(* CODESYS project CtaAppPid_2.0.0.0.library
   Description: PID Library der CTA
   Version: 2.0.0.0
   Title: CtaAppPid
   Author: SIS
   DocFormat: reStructuredText
   Placeholder: CtaAppPid
   LanguageModelAttribute: qualified-access-only
   DefaultNamespace: CtaAppPid
   CompiledLibraryCompatibilityVersion: CODESYS V3.5 SP16 Patch 3
   Company: CTA

Project tree, tasks and I/O mapping:
  libraries: CtaSysConfig, 2.0.0.0 (CTA); CtaAppTime, 1.0.0.1 (CTA); VisuSymbols, 4.5.0.0 (System); CtaVisSymbols, 2.0.0.0 (CTA); Standard, 3.5.18.0 (System); CtaAppInfluxLog, 1.0.0.1 (CTA); CtaVisHelp, 1.0.0.0 (CTA); CtaVisUser, 1.0.0.0 (CTA)
  40 Visualizations/
    visualisation popUpPID
    visualisation visPID
  30 Program Organization Units/
    function block fbPid [ST]: actConfigFile, actTrendLog, proInvert
  00000000-0000-0000-0000-000000000000|D:\CoDeSys\LibrariesV3\trunk\Intern\CAA\CAA Template\3.4.0.0 draft\Placeholder.xml
  00000000-0000-0000-0000-000000000000|D:\CoDeSys\LibrariesV3\trunk\Intern\CAA\CAA Template\3.2.0.3 draft\Prefix.pdf
  00000000-0000-0000-0000-000000000000|D:\CoDeSys\LibrariesV3\trunk\Intern\CAA\CAA Template\3.5.2.0 draft\Placeholder.xml
  20 Structs/
    data type scParameter
  50 Images/
  10 Documenation/
    global variables VersionHistory
    global variables readMe
  21 Interface/
  11 Library Parameter/
  12 Konstanten/
  60 Textlisten/
  13 Globale Variablen/
  text list GlobalTextList
*)

// 20 Structs/scParameter
TYPE scParameter :
    STRUCT
        fbrDeadBand     	:   CtaSysConfig.fbREAL;   // Dead Band
        fbrBand         	:   CtaSysConfig.fbREAL;   // Bereich in den Integriert wird in REAL
        fbrTn           	:   CtaSysConfig.fbREAL;   // Integrations Zeit in REAL 60.0 = 60.0 SEC
        fbrTv           	:   CtaSysConfig.fbREAL;   // Differential Zeit in REAL 60.0 = 60.0 SEC       
        fbxInvert			:   CtaSysConfig.fbBOOL;   // Regelverhalten Invertieren 
		fbxEnTrendlog		:	CtaSysConfig.fbBOOL;
    END_STRUCT
END_TYPE

// 10 Documenation/VersionHistory
(* 

.. image:: ../../Images/CTA_Logo.jpg
   :align: right
   :width: 15% 

**Vorlage**   


============ =========== =========== ============================================
**Date**     **Version** **Author**  **Change**
------------ ----------- ----------- --------------------------------------------
04.03.2021   0.0.0.0     SIS         Vorlage erstellt

============ =========== =========== ============================================


*)
VAR_GLOBAL
    stInfo : STRING:= '0.0.0.0, Vorlage, CTA';
END_VAR

// 10 Documenation/readMe
(*

**ReadMe**
 
 |  **Empfehlung**
 |
 |	Bibliothek CtaAppPid zur implementierung eine PID- Reglers.
 |  Instanzieren Sie den CtaAppPid.fbPid in ihrem Funktionsbaustein oder POU beispielsweise als fbPidX(Komponente)Y. (X = Nr des Reglers; Komponente z.B Pumpe, Antrieb oder Ventilator; Y = Nr der Komponente) 
 |  Deklarieren Sie die Struktur Variable welche als Parameter und zur ansteuerung dienen wie im Code beispiel.
 |  
 |  *Beispiel* 

+-----------------------+---------------------------------------------------------------------------------------------------------------------------------------------------------------------------------------------------------------------------------------------------------------------------------------------------------------------------------------------------------------------------------------------------------------------------------------+
| Beschreibung          |  Code                                                                                                                                                                                                                                                                                                                                                                                                                                 |
+=======================+=======================================================================================================================================================================================================================================================================================================================================================================================================================================+
| Pou oder SmFb         | .. code-block:: codesys                                                                                                                                                                                                                                                                                                                                                                                                               |
|                       |                                                                                                                                                                                                                                                                                                                                                                                                                                       |
|                       |	// Deklaration als VAR im POU oder dem selbsterstellten Funktionsbaustein                                                                                                                                                                                                                                                                                                                                                       	|
|                       |   VAR   																																																																																																								|
|						|	    (*PID*)																																																	 																																																						|
|						|		fbPid1Pumpe1			: CtaAppPid.fbPid;                                                                                                                                                                                                                                                                                                                                                              						|
|                       | 		fbPid2Pumpe1			: CtaAppPid.fbPid;																																																																																														|
| 						|	END_VAR                                                                                                                                                                                                                                                                                                                                                                                                                         	|
+-----------------------+---------------------------------------------------------------------------------------------------------------------------------------------------------------------------------------------------------------------------------------------------------------------------------------------------------------------------------------------------------------------------------------------------------------------------------------+
| Code für Init         | .. code-block:: codesys                                                                                                                                                                                                                                                                                                                                                                                                               |
|                       |   																																																																																																									|
| 						|	// Kopieren des nachfolgenden Codes in eine Action zur Initialisierung der Parameter. Zum Beispiel actParameter.																																																																													|
|                       |	{region "Parameter Pid1Pumpe1"}                                                                                                                                                                                                                                                                                                                                                                                                     |
| 						|		(*Basis*)																																																																																																						|
|						|		fbPid1Pumpe1.scParameter.fbrDeadBand               		(_wertInit :=   0.0									, _minInit :=   	, _maxInit := 		);		//P1 Totband																																																														|
|						|		fbPid1Pumpe1.scParameter.fbrBand						(_wertInit :=   0.0									, _minInit :=   	, _maxInit := 		);		//P2 P- Band																																																														|
|						|		fbPid1Pumpe1.scParameter.fbrTn							(_wertInit :=   0.0									, _minInit :=   	, _maxInit := 		);		//P3 Nachstellzeit																																																													|
|						|		fbPid1Pumpe1.scParameter.fbrTv							(_wertInit :=   0.0									, _minInit :=   	, _maxInit := 		);		//P4 Vorhaltezeit																																																													|
|						|		fbPid1Pumpe1.scParameter.fbxInvert						(_wertInit := FALSE																			);		//P5 Regler Invertierung																																																											|
|						|	{endregion}                                                                                                                                                      																																																																	| 
+-----------------------+---------------------------------------------------------------------------------------------------------------------------------------------------------------------------------------------------------------------------------------------------------------------------------------------------------------------------------------------------------------------------------------------------------------------------------------+
*)                                                                                                                                                                                                                                                                                                                                                                                                                                                               
 VAR_GLOBAL                                                                                                                                                                                                                                                                                                                                                                                                                                                      
    xReadMeDone              :   BOOL;                                                                                                                                                                                                                                                                                                                                                                                                                           
END_VAR

// 30 Program Organization Units/fbPid
//*******************************************************************************************************************************************************************************************************************************************//
//  Author:         SIS                                                                           																																			 //
//  Version:        1.0.0.0		                                                                      																																		 //
//  Beschreibung:   PID Regler                                                                   																																			 //
//  rIntegral =(((rAct-rSoll)/rBand*2000)/(rTn) *(rCycleTime) + rIntegral)     																										                                                	     //
//  rProp = ((rAct-rSoll)/rBand*2000)                                          																						 				                                                		 //
//  Regler Wert = ( rProp + rIntegral + rDiff)                                 																										                                                	  	 //
//*******************************************************************************************************************************************************************************************************************************************//
{attribute 'reflection'} 
FUNCTION_BLOCK fbPid 
//===========================================================================================================================================================================================================================================//
//  Variabeln Deklaration  Input                                                                  																																			 //
//===========================================================================================================================================================================================================================================//
VAR_INPUT   
    xEn                         :   BOOL;   // regler Freigabe                   
    rAct                        :   REAL;   // regelwert X in REAL
    rSoll                       :   REAL;   // Regelwert W in REAL     
    stPhysikalischeEinheit      :   STRING[5];
END_VAR
//===========================================================================================================================================================================================================================================//
//  Variabeln Deklaration  Output                                                                																																			 //
//===========================================================================================================================================================================================================================================//
VAR_OUTPUT                     
    rY              :   REAL;   // Stellgrösse Y
END_VAR
VAR
    {attribute 'instance-path'} 
    {attribute 'noinit'} 
    stInstanzName   :   STRING;
    xInitDone       :   BOOL;                                   // Inititalisierung Abgeschlossen
    scParameter     :   scParameter;
    xSimulation     :   BOOL;                                   // Simultion Aktiv
    xSimOn          :   BOOL;                                   // Simulationstrigger On
    xSimOff         :   BOOL;                                   // Simulationstrigger Off    
    rSollSim        :   REAL;                                   // Simulations Regelwert W in REAL  
    rActSim         :   REAL;                                   // Simulation Regelwert X in REAL  
    rSollPid        :   REAL;                                   // Regelwert auf den Geregelt wird
    rActPid         :   REAL;                                   // Istwert auf den Geregelt wird 
    rProp           :   REAL;                                   // Proportional Wert
    rPropVisu       :   REAL;                                   // Proportional Wert für Visu Darstellung
    rIntegral       :   REAL;                                   // Integral Wert
    rDiff           :   REAL;                                   // Diferential Wert
    xCycleStart     :	BOOL;                                   // Startbefehl des Zyklus
    xCycleInterupt  :   BOOL;                                   // Zyklus ende 
    rE              :   REAL;                                   // Aktuelle Regelabweichung
    rDeltaE         :   REAL;                                   // Regelabweichungs differenz
    rEAlt           :   REAL;                                   // Vorherergangene Regelabweichung
    rCycleTime      :	REAL;                                   // Zylkuszeit
    fbCycle         :   CtaAppTime.fbTimeMeasurement;
    fbConfigFile    :   CtaSysConfig.fbConfigFile;      		// ConfigFile Fb
    iInvert         :   INT;
    xTrigInvertPos  :   BOOL;
    xTrigInvertNeg  :   BOOL; 
(* Trendaufzeichnung *)   
    fbTrendrIst		:   CtaAppInfluxLog.FB_LOG_NODE_REAL;
    fbTrendrSoll	:   CtaAppInfluxLog.FB_LOG_NODE_REAL;
    fbTrendrY		:   CtaAppInfluxLog.FB_LOG_NODE_REAL;
END_VAR
//*******************************************************************************************************************************************************************************************************************************************//
// Upper Side must be Copied in the Var deklaration if its not possible to deklarate in the ST-Code																																			 //
//*******************************************************************************************************************************************************************************************************************************************//

//===========================================================================================================================================================================================================================================//
//  Config File                                                                                  																																			 //
//===========================================================================================================================================================================================================================================//
actConfigFile();
//===========================================================================================================================================================================================================================================//
// Sprungantwort berechnung                                                                                                                                                                                                                  //
//===========================================================================================================================================================================================================================================//
(* Regelabweichung Speichern *)
rEAlt:= rE;
// Zykluszeit erkennen
rCycleTime  :=  LTIME_TO_REAL(fbCycle.stop())/1000000000; // Ltime to ms
fbCycle.Start();

(* Freigabe *)
IF (xEn OR xSimulation) AND xInitDone AND rCycleTime > 0 THEN  
    IF xSimulation THEN
        rActPid     := rActSim;
        rSollPid    := rSollSim;
        IF NOT xSimOn THEN
            rProp       := 0;
            rIntegral   := 0;
            rDiff       := 0;
            xSimOn      := TRUE;   
            xSimOff     := FALSE;         
		END_IF;
    ELSE
        rActPid     := rAct;
        rSollPid    := rSoll;     
        IF NOT xSimOff THEN
            rProp       := 0;
            rIntegral   := 0;
            rDiff       := 0;
            xSimOff     := TRUE;   
            xSimOn      := FALSE;         
		END_IF;           
	END_IF;
    (* Invertierung *)  
    IF scParameter.fbxInvert.proValue THEN
        iInvert := -1;
        IF NOT xTrigInvertNeg THEN
            rProp       := 0;
            rIntegral   := 0;
            rDiff       := 0;
            xTrigInvertNeg := TRUE;  
            xTrigInvertPos := FALSE;   
		END_IF;
    ELSE        
        iInvert := 1;
        IF NOT xTrigInvertPos THEN
            rProp       := 0;
            rIntegral   := 0;
            rDiff       := 0;
            xTrigInvertPos := TRUE; 
            xTrigInvertNeg := FALSE;   
        END_IF;       
    END_IF;   
    // Verhinderung Division durch 0
    IF NOT(scParameter.fbrBand.proValue = 0) AND NOT xCycleStart THEN
        // Proportionalwert berechnung für Visu Dartstellung
        IF rActPid <> rSollPid THEN
            rPropVisu     := (((rActPid-rSollPid)/scParameter.fbrBand.proValue)*200)*iInvert;
        ELSE
            rPropVisu     := 0;
        END_IF;        
        // Dead Band berrechnung
        IF rActPid > rSollPid + (scParameter.fbrDeadBand.proValue/2) OR rActPid < rSollPid - (scParameter.fbrDeadBand.proValue/2) THEN
            (* Rücksetzen *)
            rProp     :=          0;    
            // Proportionalwert berechnung
            IF rActPid <> rSollPid THEN
                rProp     := (((rActPid-rSollPid)/scParameter.fbrBand.proValue)*200)*iInvert;
            END_IF;
            // Integrationswerte berechnung
            IF NOT (rProp = 0.0) AND NOT (rCycleTime = 0.0) AND NOT (scParameter.fbrTn.proValue = 0) THEN
                rIntegral :=  (rProp*(rCycleTime))/(scParameter.fbrTn.proValue)+ rIntegral;
                IF rIntegral >= 100 THEN
                    rIntegral := 100;
                END_IF;
                IF rIntegral <= -100 THEN
                    rIntegral := -100;
                END_IF;                    
            END_IF;
            // Delta der Regeldifferenz zum letzten Zyklus
            rE:= rActPid-rSollPid;
            rDeltaE:= rE - reAlt;
            IF rDeltaE <> 0 AND NOT (rCycleTime = 0.0) THEN
                rDiff:= (rDeltaE / rCycleTime * scParameter.fbrTv.proValue)*iInvert;
            ELSE
                IF rDiff > 0.1 THEN
                    rDiff := rDiff - (rDiff*0.3);
                    IF rDiff < 0 THEN
                        rDiff := 0;
					END_IF;
                ELSIF rDiff < -0.1 THEN
                    rDiff := rDiff - (rDiff*0.3); 
                    IF rDiff > 0 THEN
                        rDiff := 0;
					END_IF;                    
                ELSE
                    rDiff := 0;
                END_IF;
            END_IF;
        END_IF;
        // Ausgangswert Zusammengesetzt aus Stellwert und Integrationswert
        rY := ( rProp + rIntegral + rDiff);
    // Verhinderung Division durch 0
    ELSIF scParameter.fbrBand.proValue = 0 THEN
        rProp := 0;
        rIntegral := 0;
    ELSIF rActPid = rSollPid THEN
        rProp:= 0;
    END_IF;
    //=======================================================================================================================================================================================================================================//
    //  Überlauf verhinderung des Ausgangssignales                                                   																																		 //
    //=======================================================================================================================================================================================================================================//
    // Begrenzung des Regelwertes bei > 100
    IF rY > (100) THEN
        rY := 100;
        // Eintreten des Bandes abfangen
        IF  rProp >= 100 THEN
            rIntegral := 0;
        ELSIF rDiff = 0 THEN
            rIntegral := 100- rProp;
        END_IF;
    // Begrenzung des Regelwertes bei < -100
    ELSIF rY < (-100) THEN
        rY := -100;
        // Eintreten des Bandes abfangen
        IF  rProp <= -100 THEN
            rIntegral := 0;
        ELSIF rDiff = 0 THEN
            rIntegral := -100- rProp;
        END_IF;
    END_IF; 
ELSE
//===========================================================================================================================================================================================================================================//
// Deaktivierung der Regelwerte bei Deaktivierung                                                                                                                                                                                            //
//===========================================================================================================================================================================================================================================//
    rY          := 0;
    rProp       := 0;
    rIntegral   := 0;
END_IF;
xInitDone := TRUE;
actTrendLog();

ACTION actConfigFile:
// Aufruf fbConfigFile
fbConfigFile();
(* Aufruf der Parameter Bausteine in Fb*)
scParameter.fbrDeadBand     (_usiParaNr := 1, itfConfigFb := fbConfigFile);
scParameter.fbrBand         (_usiParaNr := 2, itfConfigFb := fbConfigFile);
scParameter.fbrTn           (_usiParaNr := 3, itfConfigFb := fbConfigFile);
scParameter.fbrTv           (_usiParaNr := 4, itfConfigFb := fbConfigFile);
scParameter.fbxInvert       (_usiParaNr := 5, itfConfigFb := fbConfigFile);
scParameter.fbxEnTrendlog	(_usiParaNr := 6, itfConfigFb := fbConfigFile);
END_ACTION

ACTION actTrendLog:
(*Istwert*)
fbTrendrIst.ENABLE		:= scParameter.fbxEnTrendlog.proValue;
fbTrendrIst.KEY			:= CONCAT(STR1 := stInstanzName, STR2 := '_rIst');
fbTrendrIst.SET_VALUE	:= rAct;

(*Sollwert*)
fbTrendrSoll.ENABLE		:= scParameter.fbxEnTrendlog.proValue;
fbTrendrSoll.KEY		:= CONCAT(STR1 := stInstanzName, STR2 := '_rSoll');
fbTrendrSoll.SET_VALUE	:= rSoll;

(*Stellwert*)
fbTrendrY.ENABLE		:= scParameter.fbxEnTrendlog.proValue;
fbTrendrY.KEY			:= CONCAT(STR1 := stInstanzName, STR2 := '_rY');
fbTrendrY.SET_VALUE		:= rY;
END_ACTION

PROPERTY proInvert : BOOL
SET
scParameter.fbxInvert.proValue := proInvert;
END_SET
GET
proInvert := scParameter.fbxInvert.proValue;
END_GET
END_PROPERTY

END_FUNCTION_BLOCK

// 40 Visualizations/popUpPID
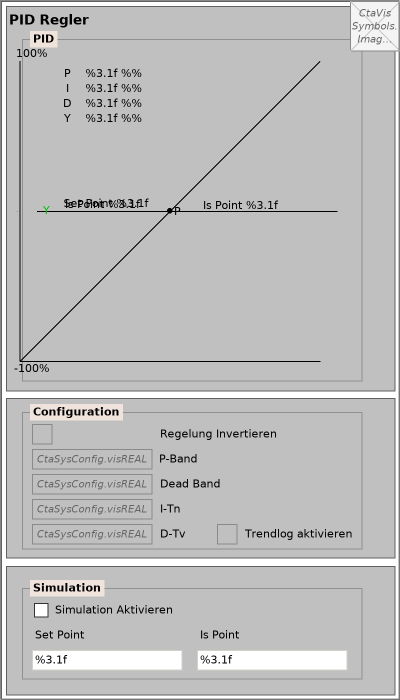
VISUALIZATION popUpPID  // 400x700
VAR_IN_OUT
    {attribute 'VAR_IN_OUT_AS_POINTER'}
    fbPID  :   fbPid;		    
END_VAR
    RoundedRectangle (1,1 399x699)
    RoundedRectangle (6,6 389x385)
    RoundedRectangle (6,398 389x160)
    RoundedRectangle (6,566 389x129)
    GroupBox (22,404 340x145), "Configuration"
        Frame (10,20 20x20)
            shows CtaSysConfig.visBOOL(visfbBOOLIn := fbPID.scParameter.fbxInvert)
        Label (135,20 150x20), "Regelung Invertieren"
        Frame (10,45 120x20)
            shows CtaSysConfig.visREAL(visfbREALIn := fbPID.scParameter.fbrBand, stPhysikalischeEinheit := fbPID.stPhysikalischeEinheit)
        Label (135,95 30x20), "I-Tn"
        Frame (10,95 120x20)
            shows CtaSysConfig.visREAL(visfbREALIn := fbPID.scParameter.fbrTn, stPhysikalischeEinheit := 's')
        Label (135,120 30x20), "D-Tv"
        Frame (10,120 120x20)
            shows CtaSysConfig.visREAL(visfbREALIn := fbPID.scParameter.fbrTv, stPhysikalischeEinheit := 's')
        Label (134,45 80x20), "P-Band"
        Frame (10,70 120x20)
            shows CtaSysConfig.visREAL(visfbREALIn := fbPID.scParameter.fbrDeadBand, stPhysikalischeEinheit := fbPID.stPhysikalischeEinheit)
        Label (135,70 80x20), "Dead Band"
        Frame (195,120 20x20)
            shows CtaSysConfig.visBOOL(visfbBOOLIn := fbPID.scParameter.fbxEnTrendlog)
        Label (220,120 115x20), "Trendlog aktivieren"
    GroupBox (22,31 340x350), "PID"
        Line (15,180) (315,180), invisible if: fbPID.scParameter.fbrDeadBand.proValue = 0.0
            p2738717112: LIMIT(-150,fbPID.scParameter.fbrDeadBand.proValue/2/MAX(0.001,fbPID.scParameter.fbrBand.proValue)*200*-1.5,150)
        Line (15,180) (315,180), invisible if: fbPID.scParameter.fbrDeadBand.proValue = 0.0
            p2738717112: LIMIT(-150,fbPID.scParameter.fbrDeadBand.proValue/2/MAX(0.001,fbPID.scParameter.fbrBand.proValue)*200*1.5,150)
        Rectangle (17,172 15x15), "Y"
    GroupBox (22,580 340x99), "Simulation"
        Textfield (10,70 150x20), "%3.1f", text variable: fbPID.rSollSim
            OnMouseDown: write the text variable via Default
        Label (10,45 150x20), "Set Point"
        Textfield (175,70 150x20), "%3.1f", text variable: fbPID.rActSim
            OnMouseDown: write the text variable via Default
        Label (175,45 150x20), "Is Point"
        Checkbox (10,20 167x20), "Simulation Aktivieren", variable: fbPID.xSimulation
    Group (10,41 310x340)
        Line (10,320) (310,20)
        Line (160,170) (160,170), invisible if: fbPID.rIntegral = 0.0
            p874137650: LIMIT(-150, TO_INT(fbPID.rProp*1.5)+TO_INT(fbPID.rIntegral*1.5),150)
            p1126004900: LIMIT(-150, - TO_INT(fbPID.rProp*1.5)-TO_INT(fbPID.rIntegral*1.5),150)
            p3528305787: LIMIT(-150, TO_INT(fbPID.rProp*1.5),150)
            p2773130477: LIMIT(-150, -TO_INT(fbPID.rProp*1.5),150)
        Line (160,170) (160,170), invisible if: fbPID.rProp = 0.0
            p874137650: LIMIT(-150, TO_INT(fbPID.rProp*1.5),150)
            p1126004900: LIMIT(-150, - TO_INT(fbPID.rProp*1.5),150)
            p3528305787: LIMIT(-150, TO_INT(fbPID.rProp*1.5),150)
        Line (160,170) (160,170), invisible if: fbPID.rProp = 0.0
            p874137650: LIMIT(-150, TO_INT(fbPID.rProp*1.5),150)
        Line (160,170) (160,170), invisible if: fbPID.rDiff = 0.0
            p874137650: LIMIT(-150, TO_INT(fbPID.rProp*1.5),150)
            p1126004900: LIMIT(-150, - TO_INT(fbPID.rProp*1.5)-TO_INT(fbPID.rDiff*1.5),150)
            p3528305787: LIMIT(-150,TO_INT(fbPID.rProp*1.5),150)
            p2773130477: LIMIT(-150,-TO_INT(fbPID.rProp*1.5),150)
        Line (10,320) (10,20)
        Line (10,320) (310,320)
        Label (0,0 44x25), "100%"
        Label (0,315 44x25), "-100%"
        Line (50,170) (160,170)
        Ellipse (157,167 5x5)
        Rectangle (49,155 98x15), "Set Point %3.1f", text variable: fbPID.rSollPid
        Ellipse (157,167 5x5)
            p3560616238: LIMIT(-150, TO_INT(fbPID.rPropVisu*1.5),150)
            p2738717112: LIMIT(-150, - TO_INT(fbPID.rPropVisu*1.5),150)
        Line (7,170) (7,170), text list: ''
            p1126004900: LIMIT(-150,-fbPID.rY*1.5,150)
        Line (160,170) (190,170), invisible if: TO_INT(fbPID.rPropVisu) > 15
            p3560616238: LIMIT(-150, TO_INT(fbPID.rPropVisu*1.5),150)
            p2738717112: LIMIT(-10, - TO_INT(fbPID.rPropVisu*1.5),150)
        Rectangle (65,25 70x15), "%3.1f %%", text variable: LIMIT(-100,fbPID.rProp,100)
        Rectangle (65,40 70x15), "%3.1f %%", text variable: LIMIT(-100, fbPID.rIntegral,100)
        Rectangle (65,55 70x15), "%3.1f %%", text variable: LIMIT(-100,fbPID.rDiff,100)
        Rectangle (50,25 15x15), "P"
        Rectangle (50,40 15x15), "I"
        Rectangle (50,55 15x15), "D"
        Rectangle (160,163 15x15), "P"
            p3560616238: LIMIT(-150, TO_INT(fbPID.rProp*1.5),150)
            p2738717112: LIMIT(-150, - TO_INT(fbPID.rProp*1.5),150)/2
        Rectangle (50,70 15x15), "Y"
        Rectangle (65,70 70x15), "%3.1f %%", text variable: LIMIT(-100,fbPID.rY,100)
        Rectangle (190,157 87x15), "Is Point %3.1f", text variable: fbPID.rActPid, invisible if: TO_INT(fbPID.rPropVisu) > 15
            p3560616238: LIMIT(-150, TO_INT(fbPID.rPropVisu*1.5),150)
            p2738717112: LIMIT(-10, - TO_INT(fbPID.rPropVisu*1.5),150)
        Group (50,156 108x15)
            Line (0,14) (108,14), invisible if: TO_INT(fbPID.rPropVisu) <= 15
                p3560616238: LIMIT(-150, TO_INT(fbPID.rPropVisu*1.5),150)
                p2738717112: LIMIT(-150, - TO_INT(fbPID.rPropVisu*1.5),150)
            Rectangle (2,0 87x15), "Is Point %3.1f", text variable: fbPID.rActPid, invisible if: TO_INT(fbPID.rPropVisu) <= 15
                p3560616238: LIMIT(-150, TO_INT(fbPID.rPropVisu*1.5),150)
                p2738717112: LIMIT(-150, - TO_INT(fbPID.rPropVisu*1.5),150)
    Image (350,1 50x50), image: CtaVisSymbols.ImagePool.close_solo_black
        OnMouseDown:  Dialog=Current Dialog, Result=OK, NumpadKeypadSet=True
    Label (6,10 150x20), "PID Regler"
    InvisibleInput (0,0 360x40)
END_VISUALIZATION

// 40 Visualizations/visPID
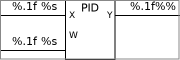
VISUALIZATION visPID  // 180x60
VAR_IN_OUT
    fbPID  :   fbPid;		
END_VAR
    Group (0,0 60x13)
        Textfield (0,0 40x13), "%.1f", text variable: fbPID.rAct
        Textfield (38,0 22x13), "%s", text variable: fbPID.stPhysikalischeEinheit
    Group (0,35 60x13)
        Textfield (0,0 40x13), "%.1f", text variable: fbPID.rSoll
        Textfield (38,0 22x13), "%s", text variable: fbPID.stPhysikalischeEinheit
    Line (0,50) (65,50)
    Line (0,15) (180,15)
    Textfield (65,0 50x60), "PID"
        OnMouseClick:  Dialog=popUpPID, Parameters={fbPID: fbPID}, Selected={0: }, OpenCentered=True
    Textfield (120,0 59x13), "%.1f%%", text variable: fbPID.rY
    Label (66,10 20x10), "X"
    Label (66,30 20x10), "W"
    Label (104,10 10x10), "Y"
END_VISUALIZATION
